FUNCTION_BLOCK Alarm
VAR_INPUT
	AlarmID : TcEventEntry;
	bRaiseAlarm : BOOL :=0;
	bConfirmAlarm : BOOL := 0;
    bClearAlarm : BOOL := 0;
	
END_VAR
VAR_OUTPUT
END_VAR
VAR
	
	bRaise : BOOL :=0;	
	bIsInitalized : BOOL :=0;
	nTimeStamp : ULINT := 0;
	fbAlarm : FB_TcALarm;
	
END_VAR

Initalize();
RaiseAlarm();
ConfirmAlarm();
ClearAlarm();
//ClearLoggedEvent();

METHOD ClearAlarm : BOOL
VAR
	bClearALL : BOOL;
END_VAR
bclearALL := MAIN.clearAlarms;
IF NOT bRaiseAlarm THEN //
	IF bClearAlarm OR bClearALL THEN	
		fbAlarm.Clear(nTimeStamp, FALSE);
	END_IF
END_IF
END_METHOD

METHOD ConfirmAlarm : BOOL
VAR_INPUT
END_VAR
IF bConfirmAlarm THEN
	fbAlarm.Confirm(nTimeStamp);
END_IF
END_METHOD

METHOD Initalize : BOOL
VAR
	fbSourceInfo : FB_TcSourceInfo;
END_VAR
IF NOT bIsInitalized THEN
	bIsInitalized := TRUE;
	//fbSourceInfo.sName := UDINT_TO_STRING(AlarmID.nEventId);
	fbAlarm.CreateEx(AlarmID, TRUE, fbSourceInfo);
END_IF
END_METHOD

METHOD RaiseAlarm : BOOL
VAR

END_VAR
bRaise := bRaiseAlarm;
IF bRaise THEN
	fbAlarm.Raise(nTimeStamp);
END_IF
END_METHOD

END_FUNCTION_BLOCK

(* stored: Version 1.1.0.1, ProductVersion 3.1.4024.6
   POU Alarm: Id {932c3d0e-2727-4df8-a543-2fcb77ec2390}, SpecialFunc None
   Method ClearAlarm: Id {e65c0889-fc79-4575-a092-b103c2499371}
   Method ConfirmAlarm: Id {1c299cc1-8493-47ab-899e-77d00fb9db6e}
   Method Initalize: Id {499d5f32-1024-45e3-9670-9fed37dd6955}
   Method RaiseAlarm: Id {e9f9ffd9-7208-4880-afdc-5e984eeac151} *)
